FUNCTION_BLOCK Test_ReadWriteBySymbolName EXTENDS TUnitTestBase
VAR
    AdsReadWriteBySymbolName : TAdsReadWriteBySymbolName;
    TestInteger : TInteger;
    ReadWriteResult : INT;    
    ScanCount : DINT;
    State: INT;
END_VAR

CASE State OF
    0:
        TestInteger.Init(1111);
        ReadWriteResult := 0;
        ScanCount := 0;
    
        AdsReadWriteBySymbolName.Execute(
            AmsNetId:= '', 
            Port:= 851, 
            SymbolName:= 'PB_TestRunner.Test_ReadWriteBySymbolName.TestInteger#Inc', 
            ReadDataAddress:= ADR(ReadWriteResult), 
            ReadDataLength:= SIZEOF(ReadWriteResult), 
            WriteDataAddress:= 0, 
            WriteDataLength:= 0, 
            KeepSymbolHandle:= FALSE);


        State := 10;
        
    10:
        ScanCount := ScanCount + 1;
        IF NOT AdsReadWriteBySymbolName.Execution.Busy THEN
            State := 20;    
		END_IF
        
    20:
        Assertion.AssertEquals_INT(
            Expected     := 1112,
            Actual       := ReadWriteResult,
            ObjectName   := _TestName,
            Variablename := 'ReadWriteResult'); 
 
        TestFinished();
        State := 0;
END_CASE

AdsReadWriteBySymbolName();

END_FUNCTION_BLOCK

(* stored: Version 1.1.0.1, ProductVersion 3.1.4024.3
   POU Test_ReadWriteBySymbolName: Id {0ffa96cd-15f2-09a0-0e25-94b697a39a97}, SpecialFunc None *)
